{attribute 'qualified_only'}
{attribute 'strict'}
TYPE E_ErrorPriority :
(
	Diagnostic := 0,
	Low := 1,
	Medium := 2,
	High := 3,
	Critical := 4
);
END_TYPE

(* stored: Version 1.1.0.1, ProductVersion 3.1.4024.12
   DUT E_ErrorPriority: Id {0898565b-041c-430c-9334-a8f65b9a52b4} *)
